// TIA Portal V16 export
// export: Created 2019-09-22T13:34:01.2045171Z, ExportSetting WithDefaults, DisplayName Totally Integrated Automation Portal, DisplayVersion V16, DisplayName TIA Portal Version Control Interface, DisplayVersion V16, DisplayName TIA Portal Openness, DisplayVersion V16, DisplayName STEP 7 Professional, DisplayVersion V16, DisplayName SIMATIC Energy Suite, DisplayVersion V16, DisplayName STEP 7 Safety, DisplayVersion V16, DisplayName WinCC Professional, DisplayVersion V16, DisplayName SIMATIC Visualization Architect, DisplayVersion V16
ORGANIZATION_BLOCK "MainDiagnostics"   // OB124, FBD, ProgramCycle
TITLE = "Main Program Sweep (Cycle)"
{ S7_Optimized_Access := 'TRUE' }
VERSION : 0.1
// //============================================================================
// //SIEMENS AG
// //(c)Copyright 2015 All Rights Reserved
// //-----------------------------------------------------------------------------
// //Library: -
// //Tested with: S7-1516-3 PN/DP FW 1.7
// //Engineering: TIA Portal V13 SP1
// //Restrictions: -
// //Requirements: -
// //Functionality: Cyclic OB for diagnostics
// //-----------------------------------------------------------------------------
// //Change log table:
// //Version  Date       Expert in charge Changes applied
// //01.00.00 24.03.2015 Siemens Industry Online Support First released version
// //============================================================================
// stored: AutoNumber true, IsIECCheckEnabled false, SetENOAutomatically false
   VAR_INPUT
      Initial_Call : Bool;   // Initial call of this OB
      Remanence : Bool;   // =True, if remanent data are available
   END_VAR
BEGIN

REGION Network 1: call function block Diagnostics
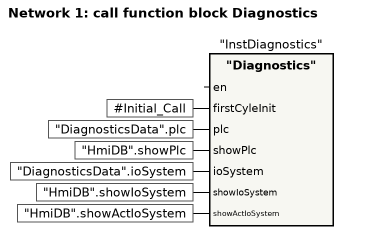
   "InstDiagnostics"(firstCyleInit := #Initial_Call,   // "Diagnostics"
                     plc := "DiagnosticsData".plc,
                     showPlc := "HmiDB".showPlc,
                     ioSystem := "DiagnosticsData".ioSystem,
                     showIoSystem := "HmiDB".showIoSystem,
                     showActIoSystem := "HmiDB".showActIoSystem);
END_REGION
END_ORGANIZATION_BLOCK
